{attribute addProperty BoxType "EJ1957-0000-0017"}
{attribute addProperty Id "FSOEAT %Q*FSOE_624AB0F2567"}
{attribute addProperty CRC "2254231546"}
{attribute addProperty SizeInBites "56"}
{attribute addProperty SizeInBytes "7"}
TYPE FSoE_Outputs_865CD7FA :
STRUCT
	{attribute addProperty Name "FSOE"}
	FSOE AT %Q* : FSOE_624AB0F2;
END_STRUCT
END_TYPE

(* stored: Version 1.2.0.0, ProductVersion 3.1.4024.9
   DUT FSoE_Outputs_865CD7FA: Id {5aba983e-2223-4ce7-a5d3-88b364544df8} *)
